PROGRAM prgHMIUnits
VAR
	tTrueUnitIndex: UINT;
	tSizeOfUnitRow: UINT;
	tSizeOfUnitRowButtons: UINT;
	tStationNumberIndexUnit: UINT;
	tScreenElementsPerPageUnit: UINT;
	tNumElementsPerScreen: UINT;
	retval: UDINT;
	nextPage: R_TRIG;
	PrevPage: R_TRIG;
END_VAR

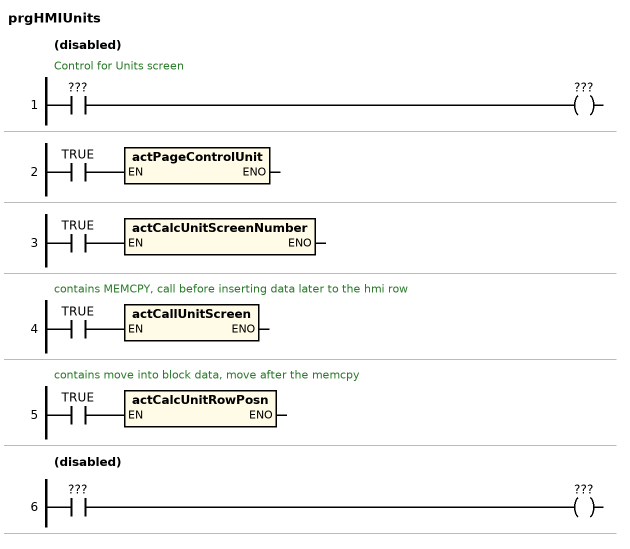
// NETWORK 1 (disabled)
// Control for Units screen
// ??? := ???;

// NETWORK 2
actPageControlUnit();

// NETWORK 3
actCalcUnitScreenNumber();

// NETWORK 4
// contains MEMCPY, call before inserting data later to the hmi row
actCallUnitScreen();

// NETWORK 5
// contains move into block data, move after the memcpy
actCalcUnitRowPosn();

// NETWORK 6 (disabled)
// ??? := ???;

ACTION actCalcUnitRowPosn:
//calculate station index for pages
tTrueUnitIndex :=	tStationNumberIndexUnit +
					(tScreenElementsPerPageUnit * gHMIUnits.gUnitActivePageNumber) -  tScreenElementsPerPageUnit;
					
//calculate offset for row x
gHMIUnits.gUnitRowElementOffset[1] :=	tTrueUnitIndex + 
										(gHMIDataConst.gNumberElementsPerRow * 1) - gHMIDataConst.gNumberElementsPerRow;

gHMIUnits.gUnitRowElementOffset[2] :=	tTrueUnitIndex + 
										(gHMIDataConst.gNumberElementsPerRow * 2) - gHMIDataConst.gNumberElementsPerRow;

gHMIUnits.gUnitRowElementOffset[3] :=	tTrueUnitIndex + 
										(gHMIDataConst.gNumberElementsPerRow * 3) - gHMIDataConst.gNumberElementsPerRow;

gHMIUnits.gUnitRowElementOffset[4] :=	tTrueUnitIndex + 
										(gHMIDataConst.gNumberElementsPerRow * 4) - gHMIDataConst.gNumberElementsPerRow;

gHMIUnits.gUnitRowElementOffset[5] :=	tTrueUnitIndex + 
										(gHMIDataConst.gNumberElementsPerRow * 5) - gHMIDataConst.gNumberElementsPerRow;

gHMIUnits.gUnitRowElementOffset[6] :=	tTrueUnitIndex + 
										(gHMIDataConst.gNumberElementsPerRow * 6) - gHMIDataConst.gNumberElementsPerRow;
				
//move to global to be picked up by each row					
gHMIUnits.gUnitRows.gMotionRow1.IndexLocation := gHMIUnits.gUnitRowElementOffset[1];
gHMIUnits.gUnitRows.gMotionRow2.IndexLocation := gHMIUnits.gUnitRowElementOffset[2];
gHMIUnits.gUnitRows.gMotionRow3.IndexLocation := gHMIUnits.gUnitRowElementOffset[3];
gHMIUnits.gUnitRows.gMotionRow4.IndexLocation := gHMIUnits.gUnitRowElementOffset[4];
gHMIUnits.gUnitRows.gMotionRow5.IndexLocation := gHMIUnits.gUnitRowElementOffset[5];
gHMIUnits.gUnitRows.gMotionRow6.IndexLocation := gHMIUnits.gUnitRowElementOffset[6];
END_ACTION

ACTION actCalcUnitScreenNumber:
//create number for station
tStationNumberIndexUnit	:= 1 * 10000; //declare math for now


//calculate number of elements per screen
tNumElementsPerScreen	:= gHMIDataConst.gNumberRowsPerPage * gHMIDataConst.gNumberElementsPerRow;

//calculate screen per page index
tScreenElementsPerPageUnit := tNumElementsPerScreen * 1; //declare math for future use
END_ACTION

ACTION actCallUnitScreen:
//calculate byte offset - motions
tSizeOfUnitRow := gHMIData.gActivePageNumber * SIZEOF(gHMIUnits.gUnitRows); //for pointer use
tSizeOfUnitRow := tSizeOfUnitRow - SIZEOF(gHMIUnits.gUnitRows);

//calculate byte offset - buttons
tSizeOfUnitRowButtons := gHMIData.gActivePageNumber * SIZEOF(gHMIUnits.gUnitButtons);
tSizeOfUnitRowButtons := tSizeOfUnitRowButtons - SIZEOF(gHMIUnits.gUnitButtons);

//move data based on station and page number
//Move feedback indicator data
//Move Button BOOL state back adr(S1_Global.MotionRow)
MEMCPY(	destAddr	:= ADR(gHMIUnits.gUnitRows),
		srcAddr		:= ADR(Mc_Global.UnitRow) + tSizeOfUnitRow,
		n			:= SIZEOF(gHMIData.gLangRows)
		);

MEMCPY(	destAddr	:= ADR(Mc_Global.UnitRowBtn) + tSizeOfUnitRowButtons,
		srcAddr		:= ADR(gHMIUnits.gUnitButtons),
		n			:= SIZEOF(gHMIUnits.gUnitButtons)
		);
END_ACTION

ACTION actPageControlUnit:
//next page
nextPage(CLK	:= gHMIButtons.btnNextPage);
IF nextPage.Q THEN
	gHMIUnits.gUnitActivePageNumber	:=	gHMIUnits.gUnitActivePageNumber + 1;
END_IF

//previous page
PrevPage(CLK	:= gHMIButtons.btnPrevPage);
IF PrevPage.Q THEN
	gHMIUnits.gUnitActivePageNumber := gHMIUnits.gUnitActivePageNumber - 1;
END_IF



//apply limits
IF gHMIUnits.gUnitActivePageNumber < 1 THEN
	gHMIUnits.gUnitActivePageNumber := 1;
END_IF
	
IF gHMIUnits.gUnitActivePageNumber > gHMIUnits.gUnitMaxPageNumber THEN
	gHMIUnits.gUnitActivePageNumber := 1;
END_IF

gHMIUnits.gUnitMaxPageNumber := Mc_Global.Data.NumberOfPages;
END_ACTION

END_PROGRAM

(* stored: Version 1.1.0.1, ProductVersion 3.1.4024.12
   POU prgHMIUnits: Id {9c8f538d-0cac-44e6-9e25-d7758a4182c4}, SpecialFunc None
   Action actCalcUnitRowPosn: Id {0ed1bd8f-f015-4a6a-985d-05d471409cfd}
   Action actCalcUnitScreenNumber: Id {b6e80cd0-cc91-4db9-8a87-842cacbe5d37}
   Action actCallUnitScreen: Id {e039fd61-b4bb-4708-9a6d-dd78cbee8b4d}
   Action actPageControlUnit: Id {a7da9a64-1712-4c8f-8f04-23c77db3b428} *)
